(* Logix 5000 project; controller AnalogIO_Shared vendor 1 type 14 code 155 rev 36.11; software revision 36.00 *)

TASK MainTask (continuous, watchdog 500 ms) : MainProgram

MODULES
   Local : vendor 1 type 14 code 155 (PointIO 0, rev 36.11)
       : 1734-IE2V (PointIO 2, rev 3.1, Input RPI 80 ms)
       : 1734-OE2V (PointIO 3, rev 3.1, Output RPI 80 ms)
      Discrete_IO : Embedded (PointIO 1, rev 36.11, Output RPI 20 ms)
END_MODULES

PROGRAM MainProgram   (* main routine MainRoutine *)
VAR
   i_AnalogVoltageInput : ALIAS FOR Local:2:I.Ch0Data;
   o_AnalogVoltageOutput : ALIAS FOR Local:3:O.Ch1Data;
END_VAR

ROUTINE MainRoutine   (* ladder *)
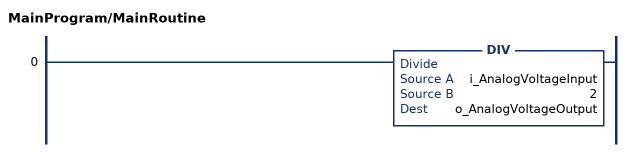
   0: DIV(i_AnalogVoltageInput,2,o_AnalogVoltageOutput);
END_ROUTINE
END_PROGRAM
